// TIA Portal V20 export
DATA_BLOCK "DB_Powermeter"   // DB433
// stored: AutoNumber false, InstanceOfName FB_Powermeter, InstanceOfType FB
"FB_Powermeter"
   // VAR
   //    sPowerMeterWorkPos : Bool;
   //    sPowerMeterHomePos : Bool;
   //    sPowerMeterToWorkMoveReq : Bool;
   //    sPowerMeterToHomeMoveReq : Bool;
   //    sPowerMeterJogMode : Bool;
   //    sPowermeterCylinder : "FB_CmdCylinder";
   //    sPowermeterInHomePos { S7_SetPoint := 'True'} : Bool;
   //    sPowermeterInMiddlePos : Bool;
   //    sPowermeterInWorkPos : Bool;
   //    sPowerMeterCylErrorCode : Int;
   //    sPowerMeterHomePosCtrlTimer : TON_TIME;
   //    sPowerMeterWorkPosCtrlTimer : TON_TIME;
   //    sMeasurePowerLaser { S7_SetPoint := 'True'} : Bool;
   //    sRTLaserMeasureON : R_TRIG;
   //    sLaserPowerValue { S7_SetPoint := 'True'} : Real;
   //    sWeightFactor : Real;
   //    sAlpha : Real;
   //    sDateAndTime : DTL;
   //    sActualMeasPower : Real;
   //    sTolMin : Real;
   //    sTolMax : Real;
   //    sResetMeasures : Bool;
   //    sPowerMeterSeq : "FB_PowerMeterSeq";
   //    RT_StartArchive { S7_SetPoint := 'True'} : R_TRIG;
   //    sArchivePmValues { S7_SetPoint := 'True'} : Array[0..4] of Real;
   // END_VAR
BEGIN
END_DATA_BLOCK
